Fanuc KAREL source: kt00129.KL

-- PROVISIONAL review KL for V770-1; original PC SHA256 dc8f6c10c2ce2973fa6802767079c6b31a518e25f94840637f1a9a229081733f
-- Incomplete behavior may be omitted. Consult companion uncertainty JSON. Do not deploy.
PROGRAM KT00129
%NOLOCKGROUP
VAR
  I1 : INTEGER
  I2 : INTEGER
  OUT : INTEGER
BEGIN
  -- UNRESOLVED_PC offsets 5-16; opcodes 2E,23
  -- UNRESOLVED_PC offsets 21-32; opcodes 2E,23
  -- UNRESOLVED_PC offsets 37-48; opcodes 2E,23
  -- UNRESOLVED_PC offsets 53-64; opcodes 2E,23
  -- UNRESOLVED_PC offsets 69-88; opcodes 21,21,55,23
  -- UNRESOLVED_PC offsets 93-97; opcodes 7F
END KT00129
